# EPICS IOC start-up script: ioc_rotary_encoder/iocBoot/iocRotaryEncoder/st.cmd.iocsh
< envPaths

epicsEnvSet("ENGINEER", "rpi")
epicsEnvSet("IOC", "iocRotaryEncoder")
epicsEnvSet("P", "RE:")
epicsEnvSet("R", "ch0:")
epicsEnvSet("SERIAL_PORT", "/dev/ttyACM0")
epicsEnvSet("SERIAL_BAUD", "115200")

cd "${TOP}"

dbLoadDatabase "dbd/RotaryEncoder.dbd"
RotaryEncoder_registerRecordDeviceDriver pdbbase

dbLoadRecords "db/RotaryEncoder.db", "P=$(P),R=$(R)"
dbl > pvlist.txt

cd "${TOP}/iocBoot/${IOC}"

iocInit

rotaryStartSerialReader("$(P)$(R)", "$(SERIAL_PORT)", "$(SERIAL_BAUD)")
